Fanuc KAREL source: TRUNC.kl

PROGRAM T
%NOLOCKGROUP
VAR
 v0 : REAL
 res : INTEGER
BEGIN
 res = TRUNC(v0)
END T
